SUBAPPLICATION Ventilsteuerung_Uebung_053 (* DigitalInput_I1-_I4 auf DigitalOutput_Q1-_Q4 *)
  (* Standard: 61499-2 *)
  (* Version 1.0, 2023-10-23, franz *)
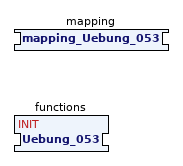
  SUBAPPS
    mapping : mapping_Uebung_053;
    functions : Uebung_053;
  END_SUBAPPS
END_SUBAPPLICATION
